# B&R Automation Studio project mappDatabase
Automation Studio 4.9.5.36 SP; technology packages: mapp 5.16.1, mappView 5.16.1

## Configuration Config1

CPU PC_any, AutomationRuntime E4.90, Build 4.1.2, Safety 0.0, Vc V4.45.0

### Task classes (Cpu.sw)
```
Cyclic#1 (cycle 10000 us):
  mappDB <- mappDatabase.mappDB.prg
  RecipeSamp <- mappDatabase.RecipeSample.prg
Binaries: mvLoader, udbdef, arsvcreg, TCData, arconfig, User, Role, Config, iomap, asfw, ashwac, ashwd, sysconf
Libraries: MpDatabase, MpBase, AsHttp, runtime, MpCom, AsBrStr, astime, arssl, asieccon, fileio, standard, IecCheck, sys_lib
```

### Hardware
```
PC : PC_any v1.1.1.0 (OrderNumber=PC)
  ConfigurationID = mappViewSample_Config1
  Cyclic1Duration = 10000
  FileDevice1
  FileDeviceName1 = MpCfgDev
  FileDevicePath1 = C:\Temp
  ActivateOpcUa = 1
  OpcUaInformationModels_PV_Version = 1
```

### Config.mpdatabasecore - PC/mappServices/Config.mpdatabasecore
```
Element gDatabaseCore (Type=mpdatabasecore)
  mapp.Database.Core:
    Name = BrDatabase
    UserName = br
    Password = bandr
    IPAddress  // IPv4 address of the database script
    PortNumber = 85  // SQL port number of the database script
    DBQueries:
      [0]:
        Name = RecipeLoad
        Type:
          Select:
            Columns:
              PV = ::Recipe.DATA
          From = dbo.BrTable
          Where:
            [0]:
              Column = product_name
              Operator = eq
              CompareTo:
                Value = {&pv[Recipe.PAR.RecipeName]}
      [1]:
        Name = RecipeSave
        Type = UPDATE
          TableName = dbo.BrTable
          Columns:
            PV = ::Recipe.DATA
          Where:
            [0]:
              Column = product_name
              Operator = eq
              CompareTo:
                Value = {&pv[Recipe.PAR.RecipeName]}
      [2]:
        Name = RecipeDelete
        Type = DELETE
          TableName = dbo.BrTable
          Where:
            [0]:
              Column = product_name
              Operator = eq
              CompareTo:
                Value = {&pv[Recipe.PAR.RecipeName]}
      [3]:
        Name = RecipeNew
        Type = INSERT
          Into = dbo.BrTable
          Columns:
            PV = ::Recipe.DATA
      [4]:
        Name = RecipeList
        Type = Custom
          Query = SELECT product_name FROM dbo.BrTable WHERE product_name LIKE '%'
          Columns = SingleColumns
            [0]:
              Column = product_name
              PV = ::Recipe.PAR.RecipeName
```

## Logical view

Binary libraries used (declarations not repeated): operator, runtime, astime, AsIecCon, AsHttp, AsBrStr, standard, IecCheck, sys_lib, FileIO, AsICMP, MpCom 5.14.1, MpBase, MpDatabase 5.16.1

### Package Logical/Libraries - Global libraries

### Library Logical/Libraries/MpCfg (IEC)

#### Types.typ - Exported data types
```iecst
TYPE
	MpCfgInfoType : 	STRUCT
		state : MpCfgStateType;
		DevLink_1 : DevLink;
		FileOpen_1 : FileOpen;
		FileRead_1 : FileRead;
		FileWrite_1 : FileWrite;
		FileClose_1 : FileClose;
		MpComConfigManager_1 : MpComConfigManager;
		Buffer : ARRAY[0..MpCfgMaxBufferSize]OF USINT;
		DataOffset1 : DINT;
		DataOffset2 : DINT;
		DataOffset3 : DINT;
		DataLen : DINT;
		FileLen : DINT;
		tmpStr1 : STRING[MpCfgMaxNameSize];
		tmpStr2 : STRING[MpCfgMaxNameSize];
		idx : UDINT;
	END_STRUCT;
	MpCfgStateType :
		(
		stateWait,
		stateDevLink,
		stateExport,
		stateOpen,
		stateRead,
		stateWrite,
		stateClose,
		stateFindGroup,
		stateFindData,
		stateInsertData,
		stateImport,
		stateError
		);
	MpCfgGroupArray : 	STRUCT
		Item : ARRAY[0..9]OF STRING[MpCfgMaxNameSize];
	END_STRUCT;
END_TYPE
```

#### Constants.var - Exported constants
```iecst
(*Buffer and variable sizes*)
VAR CONSTANT
	MpCfgMaxBufferSize : UINT := 20000; (*Maximum size of the configuration file*)
	MpCfgMaxNameSize : UINT := 200; (*Maximum length of the parameter name*)
	MpCfgMaxValueSize : UINT := 200; (*Maximum length of the value information*)
END_VAR
(*Error numbers*)
VAR CONSTANT
	MpCfgBufferSizeExceeded : DINT := 10001; (*Configuration file is larger than MpCfgMaxBufferSize | Increase value of MpCfgMaxBufferSize*)
	MpCfgDataTypeSizeExceeded : DINT := 10002; (*Data type information is larger than MpCfgMaxNameSize | Increase value of MpCfgMaxNameSize*)
	MpCfgValueSizeExceeded : DINT := 10003; (*Value length is larger than MpCfgMaxNameSize | Increase value of MpCfgMaxNameSize*)
	MpCfgGroupNotFound0 : DINT := 10010; (*Group name does not exist | Check group array data at index x*)
	MpCfgGroupNotFound1 : DINT := 10011; (*Group name does not exist | Check group array data at index x*)
	MpCfgGroupNotFound2 : DINT := 10012; (*Group name does not exist | Check group array data at index x*)
	MpCfgGroupNotFound3 : DINT := 10013; (*Group name does not exist | Check group array data at index x*)
	MpCfgGroupNotFound4 : DINT := 10014; (*Group name does not exist | Check group array data at index x*)
	MpCfgGroupNotFound5 : DINT := 10015; (*Group name does not exist | Check group array data at index x*)
	MpCfgGroupNotFound6 : DINT := 10016; (*Group name does not exist | Check group array data at index x*)
	MpCfgGroupNotFound7 : DINT := 10017; (*Group name does not exist | Check group array data at index x*)
	MpCfgGroupNotFound8 : DINT := 10018; (*Group name does not exist | Check group array data at index x*)
	MpCfgGroupNotFound9 : DINT := 10019; (*Group name does not exist | Check group array data at index x*)
	MpCfgParaNotFound : DINT := 10020; (*Parameter name does not exist in configuration | Double check parameter name*)
	MpCfgTypeNotFound : DINT := 10021; (*Data type information was not found | Shouldnt happen but just in case it does*)
	MpCfgValueNotFound : DINT := 10022; (*Value information was not found | Shouldnt happen but just in case it does*)
	MpCfgParaNameEmpty : DINT := 10030; (*Parameter name is empty*)
	MpCfgMpLinkEmpty : DINT := 10031; (*mapp Link is missing*)
END_VAR
(*Read/Write constants*)
VAR CONSTANT
	MpCfgRead : BOOL := FALSE;
	MpCfgWrite : BOOL := TRUE;
END_VAR
```

#### MpCfg.fun - Exported functions and function blocks
```iecst
FUNCTION_BLOCK MpCfgRW
	VAR_INPUT
		MpLink : {REDUND_UNREPLICABLE} MpComIdentType;
		Enable : BOOL;
		ReadWrite : BOOL;
		ErrorReset : BOOL;
		ParaName : STRING[MpCfgMaxNameSize];
		ParaValue : STRING[MpCfgMaxValueSize];
		GroupArray : REFERENCE TO MpCfgGroupArray;
	END_VAR
	VAR_OUTPUT
		Active : BOOL;
		Error : BOOL;
		StatusID : DINT;
		CommandDone : BOOL;
		DataType : STRING[50];
		Value : STRING[MpCfgMaxValueSize];
	END_VAR
	VAR
		Info : MpCfgInfoType;
		zzEdge00000 : BOOL;
		zzEdge00001 : BOOL;
	END_VAR
END_FUNCTION_BLOCK

FUNCTION FindInMem : DINT
	VAR_INPUT
		data1 : UDINT;
		len1 : UDINT;
		data2 : UDINT;
		len2 : UDINT;
		direction : BOOL;
	END_VAR
	VAR
		idx : UDINT;
	END_VAR
END_FUNCTION
```

#### MpCfg.st
```iecst
// -------------------------------------------------------------------------
// Read mapp configuration parameter
// -------------------------------------------------------------------------
FUNCTION_BLOCK MpCfgRW
	// Abort command
	IF EDGENEG(Enable) THEN
		// Close file if it was already opened
		IF Info.state >= stateOpen AND Info.state <> stateError THEN
			Info.state := stateClose;
		END_IF
	END_IF

	// -------------------------------------------------------------------------
	// MpLink state machine
	CASE Info.state OF
		// -------------------------------------------------------------------------
		// Wait for new command
		stateWait:
			// Reset all funtion blocks
			Info.DevLink_1.enable 				:= FALSE;
			Info.DevLink_1();
			Info.MpComConfigManager_1.Enable 	:= FALSE;
			Info.MpComConfigManager_1();
			Info.FileOpen_1.enable				:= FALSE;
			Info.FileOpen_1();
			Info.FileRead_1.enable				:= FALSE;
			Info.FileRead_1();
			Info.FileClose_1.enable				:= FALSE;
			Info.FileClose_1();

			// New command
			IF EDGEPOS(Enable) THEN
				// Make sure MpLink is not empty
				IF MpLink.Internal[0] = 0 THEN
					StatusID := MpCfgMpLinkEmpty;
					Info.state := stateError;
				ELSE
					// Make sure parameter is not empty
					IF ParaName = '' THEN
						StatusID := MpCfgParaNameEmpty;
						Info.state := stateError;
					ELSE
						// Set start values
						Active := TRUE;
						DataType := '';
						Value := '';
						brsmemset(ADR(Info.Buffer), 0, SIZEOF(Info.Buffer));
						Info.state := stateDevLink;
					END_IF
				END_IF
			ELSE
				IF NOT Enable THEN
					CommandDone := FALSE;
				END_IF
				Active := FALSE;
			END_IF
			// -------------------------------------------------------------------------
		// Link file device used for exporting data
		stateDevLink:
			Info.DevLink_1.enable 	:= TRUE;
			Info.DevLink_1.pDevice	:= ADR('MpCfgDev');
			Info.DevLink_1.pParam	:= ADR('/DEVICE=C:/');
			Info.DevLink_1();

			// Success
			IF Info.DevLink_1.status = ERR_OK OR Info.DevLink_1.status = fiERR_DEVICE_ALREADY_EXIST THEN
				Info.state := stateExport;
			// Errror
			ELSIF Info.DevLink_1.status <> ERR_FUB_BUSY THEN
				StatusID := Info.DevLink_1.status;
				Info.state := stateError;
			END_IF
		// -------------------------------------------------------------------------
		// Export mapp data
		stateExport:
			Info.MpComConfigManager_1.Enable 		:= TRUE;
			Info.MpComConfigManager_1.MpLink		:= ADR(MpLink);
			Info.MpComConfigManager_1.DeviceName 	:= ADR('MpCfgDev');
			Info.MpComConfigManager_1.FileName 		:= ADR('MpCfg.xml');
			Info.MpComConfigManager_1.Scope			:= mpCOM_CONFIG_SCOPE_COMPONENT;
			Info.MpComConfigManager_1.Export		:= TRUE;
			Info.MpComConfigManager_1.Import		:= FALSE;
			Info.MpComConfigManager_1();

			// Success
			IF Info.MpComConfigManager_1.CommandDone AND NOT Info.MpComConfigManager_1.Error THEN
				Info.state := stateOpen;
			// Errror
			ELSIF Info.MpComConfigManager_1.Error THEN
				StatusID := Info.MpComConfigManager_1.StatusID;
				Info.state := stateError;
			END_IF
		// -------------------------------------------------------------------------
		// Open mapp data
		stateOpen:
			Info.FileOpen_1.enable		:= TRUE;
			Info.FileOpen_1.pDevice 	:= ADR('MpCfgDev');
			Info.FileOpen_1.pFile		:= ADR('MpCfg.xml');
			Info.FileOpen_1.mode 		:= fiREAD_WRITE;
			Info.FileOpen_1();

			// Success
			IF Info.FileOpen_1.status = ERR_OK THEN
				IF Info.FileOpen_1.filelen > SIZEOF(Info.Buffer) THEN
					StatusID := MpCfgBufferSizeExceeded;
					Info.state := stateError;
				ELSE
					Info.state := stateRead;
				END_IF
			// Errror
			ELSIF Info.FileOpen_1.status <> ERR_FUB_BUSY THEN
				StatusID := Info.FileOpen_1.status;
				Info.state := stateError;
			END_IF

		// -------------------------------------------------------------------------
		// Read mapp data file
		stateRead:
			Info.FileRead_1.enable		:= TRUE;
			Info.FileRead_1.ident		:= Info.FileOpen_1.ident;
			Info.FileRead_1.len			:= Info.FileOpen_1.filelen;
			Info.FileRead_1.pDest		:= ADR(Info.Buffer);
			Info.FileRead_1();

			// Success
			IF Info.FileRead_1.status = ERR_OK THEN
				Info.idx := 0;
				Info.DataOffset1 := 0;
				// Find group id first
				IF ADR(GroupArray) <> 0 THEN
					// Make sure array has at least one entry
					IF GroupArray.Item[0] <> '' THEN
						Info.state := stateFindGroup;
					// Find unique parameter
					ELSE
						Info.state := stateFindData;
					END_IF
				// Find unique parameter
				ELSE
					Info.state := stateFindData;
				END_IF
			// Errror
			ELSIF Info.FileRead_1.status <> ERR_FUB_BUSY THEN
				StatusID := Info.FileRead_1.status;
				Info.state := stateError;
			END_IF

		// -------------------------------------------------------------------------
		// Write mapp data file
		stateWrite:
			Info.FileWrite_1.enable		:= TRUE;
			Info.FileWrite_1.ident		:= Info.FileOpen_1.ident;
			Info.FileWrite_1.len		:= Info.FileLen;
			Info.FileWrite_1.pSrc		:= ADR(Info.Buffer);
			Info.FileWrite_1();

			// Success
			IF Info.FileWrite_1.status = ERR_OK THEN
				Info.state := stateClose;
			// Errror
			ELSIF Info.FileWrite_1.status <> ERR_FUB_BUSY THEN
				StatusID := Info.FileWrite_1.status;
				Info.state := stateError;
			END_IF

		// -------------------------------------------------------------------------
		// Find group data
		stateFindGroup:
			// Prepare group string
			Info.tmpStr1 := '<Group ID="';
			brsstrcat(ADR(Info.tmpStr1), ADR(GroupArray.Item[Info.idx]));
			brsstrcat(ADR(Info.tmpStr1), ADR('"'));
			// Find property string
			Info.DataOffset1 := Info.DataOffset1+FindInMem(ADR(Info.Buffer)+Info.DataOffset1, Info.FileOpen_1.filelen, ADR(Info.tmpStr1), brsstrlen(ADR(Info.tmpStr1)), FALSE);

			// Found group string
			IF Info.DataOffset1 > -1 THEN
				// Find next group name
				IF Info.idx < SIZEOF(GroupArray)/SIZEOF(GroupArray.Item[0]) THEN
					Info.idx := Info.idx + 1;
					IF GroupArray.Item[Info.idx] = '' THEN
						Info.state := stateFindData;
					END_IF
				// Group was not found
				ELSE
					StatusID := MpCfgGroupNotFound0+Info.idx;
					Info.state := stateError;
				END_IF
			// Group was not found
			ELSE
				StatusID := MpCfgGroupNotFound0+Info.idx;
				Info.state := stateError;
			END_IF
		// -------------------------------------------------------------------------
		// Find data
		stateFindData:
			// Prepare property string
			Info.tmpStr1 := '<Property ID="';
			brsstrcat(ADR(Info.tmpStr1), ADR(ParaName));
			brsstrcat(ADR(Info.tmpStr1), ADR('"'));
			// Find property string
			Info.DataOffset2 := FindInMem(ADR(Info.Buffer)+Info.DataOffset1, Info.FileOpen_1.filelen, ADR(Info.tmpStr1), brsstrlen(ADR(Info.tmpStr1)), FALSE);

			// Found parameter string
			IF Info.DataOffset2 > -1 THEN
				Info.DataOffset1 := Info.DataOffset1+Info.DataOffset2;
				// Prepare data type start string
				Info.tmpStr1 := 'DataType="';
				// Find data type string start
				Info.DataOffset2 := brsstrlen(ADR(Info.tmpStr1))+FindInMem(ADR(Info.Buffer)+Info.DataOffset1, Info.FileOpen_1.filelen, ADR(Info.tmpStr1), brsstrlen(ADR(Info.tmpStr1)), FALSE);

				// Found data type start
				IF Info.DataOffset2 > -1 THEN
					// Prepare data type end string
					Info.tmpStr1 := '"';
					// Find data type string
					Info.DataLen := FindInMem(ADR(Info.Buffer)+Info.DataOffset1+Info.DataOffset2, Info.FileOpen_1.filelen, ADR(Info.tmpStr1), brsstrlen(ADR(Info.tmpStr1)), FALSE);

					// Found data type end, copy data to output
					IF Info.DataLen > -1 THEN
						brsmemset(ADR(DataType), 0, SIZEOF(DataType));
						brsmemcpy(ADR(DataType), ADR(Info.Buffer)+Info.DataOffset1+Info.DataOffset2, Info.DataLen);

						// Prepare value start string
						Info.tmpStr1 := 'Value="';
						// Find data type string start
						Info.DataOffset2 := brsstrlen(ADR(Info.tmpStr1))+FindInMem(ADR(Info.Buffer)+Info.DataOffset1, Info.FileOpen_1.filelen, ADR(Info.tmpStr1), brsstrlen(ADR(Info.tmpStr1)), FALSE);

						// Found value start
						IF Info.DataOffset2 > -1 THEN
							// Prepare value end string
							Info.tmpStr1 := '"';
							// Find value end string
							Info.DataLen := FindInMem(ADR(Info.Buffer)+Info.DataOffset1+Info.DataOffset2, Info.FileOpen_1.filelen, ADR(Info.tmpStr1), brsstrlen(ADR(Info.tmpStr1)), FALSE);

							// Found value end, copy data to output
							IF Info.DataLen > -1 THEN
								brsmemset(ADR(Value), 0, SIZEOF(Value));
								brsmemcpy(ADR(Value), ADR(Info.Buffer)+Info.DataOffset1+Info.DataOffset2, Info.DataLen);

								// Finish when command is reading
								IF ReadWrite = MpCfgRead THEN
									Info.state := stateClose;
								// Insert new data in next step
								ELSE
									Info.state := stateInsertData;
								END_IF
							// Value end was not found
							ELSE
								StatusID := MpCfgValueNotFound;
								Info.state := stateError;
							END_IF
						// Value start was not found
						ELSE
							StatusID := MpCfgValueNotFound;
							Info.state := stateError;
						END_IF
					// Data type end was not found
					ELSE
						StatusID := MpCfgTypeNotFound;
						Info.state := stateError;
					END_IF
				// Data type end was not found
				ELSE
					StatusID := MpCfgTypeNotFound;
					Info.state := stateError;
				END_IF
			// Parameter name was not found
			ELSE
				StatusID := MpCfgParaNotFound;
				Info.state := stateError;
			END_IF

		// -------------------------------------------------------------------------
		// Insert new data
		stateInsertData:
			// Calculate start address for value
			Info.DataOffset3 := ADR(Info.Buffer)+Info.DataOffset1+Info.DataOffset2;
			// Calculate remaining data
			Info.DataLen := Info.FileOpen_1.filelen-(Info.DataOffset1+Info.DataOffset2);

			brsmemmove(Info.DataOffset3+brsstrlen(ADR(ParaValue)), Info.DataOffset3+brsstrlen(ADR(Value)), Info.DataLen-brsstrlen(ADR(Value))+1);
			brsmemcpy(Info.DataOffset3, ADR(ParaValue), brsstrlen(ADR(ParaValue)));

			// New value is shorter than old
			IF brsstrlen(ADR(Value)) >= brsstrlen(ADR(ParaValue)) THEN
				Info.FileLen := Info.FileOpen_1.filelen;
				// Fill taling memory with LF if new data is smaller than old
				brsmemset(ADR(Info.Buffer)+Info.FileLen, 10, brsstrlen(ADR(Value))-brsstrlen(ADR(ParaValue)));
			// New value is larger than old
			ELSE
				Info.FileLen := Info.FileOpen_1.filelen+(brsstrlen(ADR(ParaValue))-brsstrlen(ADR(Value)));
			END_IF

			Info.state := stateWrite;

		// -------------------------------------------------------------------------
		// Close mapp data file
		stateClose:
			Info.FileClose_1.enable		:= TRUE;
			Info.FileClose_1.ident		:= Info.FileOpen_1.ident;
			Info.FileClose_1();

			// Success
			IF Info.FileClose_1.status = ERR_OK THEN
				Info.FileOpen_1.enable := FALSE;

				// When we read it ends here
				IF ReadWrite = MpCfgRead THEN
					Active := FALSE;
					CommandDone := TRUE;
					Info.state := stateWait;
				// Import new configuration
				ELSE
					Info.state := stateImport;
				END_IF
				// Errror
			ELSIF Info.FileClose_1.status <> ERR_FUB_BUSY THEN
				StatusID := Info.FileClose_1.status;
				Info.state := stateError;
			END_IF

		// -------------------------------------------------------------------------
		// Import mapp data
		stateImport:
			Info.MpComConfigManager_1.Enable 		:= TRUE;
			Info.MpComConfigManager_1.MpLink		:= ADR(MpLink);
			Info.MpComConfigManager_1.DeviceName 	:= ADR('MpCfgDev');
			Info.MpComConfigManager_1.FileName 		:= ADR('MpCfg.xml');
			Info.MpComConfigManager_1.Scope			:= mpCOM_CONFIG_SCOPE_COMPONENT;
			Info.MpComConfigManager_1.Export		:= FALSE;
			Info.MpComConfigManager_1.Import		:= TRUE;
			Info.MpComConfigManager_1();

			// Success
			IF Info.MpComConfigManager_1.CommandDone AND NOT Info.MpComConfigManager_1.Error THEN
				Active := FALSE;
				CommandDone := TRUE;
				Info.state := stateWait;
			// Errror
			ELSIF Info.MpComConfigManager_1.Error THEN
				StatusID := Info.MpComConfigManager_1.StatusID;
				Info.state := stateError;
			END_IF

		// -------------------------------------------------------------------------
		// Error state
		stateError:
			// Close file when it is open
			IF Info.FileOpen_1.enable THEN
				Info.FileClose_1.enable	:= TRUE;
				Info.FileClose_1.ident	:= Info.FileOpen_1.ident;
				Info.FileClose_1();
			END_IF

			// Set flags
			Active := FALSE;
			Error := TRUE;
			CommandDone := TRUE;

			// Wait for error reset
			IF ErrorReset THEN
				StatusID := 0;
				Error := FALSE;
				Info.state := stateWait;
			END_IF
	END_CASE;

	ErrorReset := FALSE;
END_FUNCTION_BLOCK
```

#### LocalFunctions.st
```iecst
//******************************************************************************************************
// Find second data in first data
//******************************************************************************************************
FUNCTION FindInMem
	FindInMem := -1;
	IF (len1 > len2) THEN
		IF(direction) THEN
			idx := len1 - len2;
			WHILE(idx > 0) DO
				IF (brsmemcmp(data1 + idx, data2, len2) = 0) THEN
					FindInMem := idx;
					EXIT;
				END_IF
				idx := idx - 1;
			END_WHILE;
		ELSE
			FOR idx:=0 TO len1 - len2 DO
				IF (brsmemcmp(data1 + idx, data2, len2) = 0) THEN
					FindInMem := idx;
					EXIT;
				END_IF
			END_FOR;
		END_IF
	END_IF
END_FUNCTION
```

#### changelog.txt
```
Version 1.0 (23.12.2021)
- First public release
```

- Visualisation Logical/mappView (not shown)

### Program Logical/mappDatabase/mappDB (IEC)

#### Main.st - Init, cyclic, exit code
```iecst
PROGRAM _INIT
	// --------------------------------------------------------------------------------------------------------------------
	// Preset function blocks
	MpDatabaseCore_0.MpLink := ADR(gDatabaseCore);
	MpDatabaseQuery_0.MpLink := ADR(gDatabaseCore);

	SqlTimeout.PT := TIMEOUT;

	REPEAT
		MpCfgRW_01.Enable 		:= TRUE;
		MpCfgRW_01.MpLink 		:= gDatabaseCore;
		MpCfgRW_01.ReadWrite 	:= MpCfgRead;
		MpCfgRW_01.ParaName 	:= 'IPAddress';
		MpCfgRW_01.GroupArray	:= 0;
		MpCfgRW_01();
		UNTIL MpCfgRW_01.CommandDone
	END_REPEAT;

END_PROGRAM

PROGRAM _CYCLIC
		// Trigger ping request
	PingTimer.IN := TRUE;
	PingTimer.PT := PING_TIMEOUT;
	PingTimer();
	// Try to ping network share if not connected
	IF(MpCfgRW_01.Value <> '' AND PingTimer.Q) THEN
		IcmpPing_0(enable := 1, pHost := ADR(MpCfgRW_01.Value), timeout := PING_TIMEOUT);
		// Ping was OK
		IF(IcmpPing_0.status = ERR_OK) THEN
			PingTimer(IN := FALSE);
			Database.PAR.CanPing := TRUE;
			// Disconnect from share when ping failed
		ELSIF(IcmpPing_0.status <> ERR_FUB_BUSY) THEN
			PingTimer(IN := FALSE);
			Database.PAR.CanPing := FALSE;
			IF(Database.PAR.IsConnected) THEN
				Database.CMD.Disconnect := TRUE;
			END_IF
		END_IF
	ELSIF(PingTimer.Q) THEN
		PingTimer(IN := FALSE);
	END_IF

	// --------------------------------------------------------------------------------------------------------------------
	// Database state machine
	// --------------------------------------------------------------------------------------------------------------------
	CASE dbState OF
		// --------------------------------------------------------------------------------------------------------------------
		// Wait state
		dbSTATE_WAIT:
			// --------------------------------------------------------------------------------------------------------------------
			// Connect to database
			IF Database.CMD.Connect THEN
				dbState := dbSTATE_CONNECT;
			END_IF

			// Disconnect from database
			IF Database.CMD.Disconnect THEN
				dbState := dbSTATE_DISCONNECT;
			END_IF

			// Execute SQL command
			IF Database.CMD.Execute THEN
				dbState := dbSTATE_QUERY;
			END_IF

			// Get next entry
			IF Database.CMD.NextRow THEN
				dbState := dbSTATE_NEXT;
			END_IF

			// --------------------------------------------------------------------------------------------------------------------
			// Reset error information and timeout timer
			IF Database.CMD.Connect OR Database.CMD.Disconnect OR Database.CMD.Execute OR Database.CMD.NextRow THEN
				Database.ERR.No := 0;
				brsmemset(ADR(Database.ERR.Text), 0, SIZEOF(Database.ERR.Text));

				MpDatabaseCore_0.Enable := TRUE;
				MpDatabaseQuery_0.Enable := TRUE;
				MpDatabaseQuery_0.ErrorReset := TRUE;
				MpDatabaseCore_0.ErrorReset := TRUE;
				MpDatabaseQuery_0();
				MpDatabaseCore_0();

				SqlTimeout.IN := 0;
				SqlTimeout();
			END_IF

		// --------------------------------------------------------------------------------------------------------------------
		// Connect state
		dbSTATE_CONNECT:
			SqlTimeout.IN := 1;
			SqlTimeout();

			IF MpDatabaseCore_0.CommandDone OR MpDatabaseCore_0.Error THEN
				IF MpDatabaseCore_0.Error THEN
					Database.ERR.No := MpDatabaseCore_0.StatusID;
					dbState := dbSTATE_ERROR;
				ELSE
					Database.CMD.Connect := FALSE;
					dbState := dbSTATE_WAIT;
				END_IF
			ELSIF SqlTimeout.Q THEN
				Database.ERR.No := ERR_SQL_TIMEOUT_CONNECT;
				MpDatabaseCore_0.Enable := FALSE;
				dbState := dbSTATE_ERROR;
			END_IF

		// --------------------------------------------------------------------------------------------------------------------
		// Disconnect state
		dbSTATE_DISCONNECT:
			SqlTimeout.IN := 1;
			SqlTimeout();

			IF MpDatabaseCore_0.CommandDone OR MpDatabaseCore_0.Error THEN

				IF MpDatabaseCore_0.Error THEN
					Database.ERR.No := MpDatabaseCore_0.StatusID;
					dbState := dbSTATE_ERROR;
				ELSE
					Database.CMD.Disconnect := FALSE;
					dbState := dbSTATE_WAIT;
				END_IF
			ELSIF SqlTimeout.Q THEN
				Database.ERR.No := ERR_SQL_TIMEOUT_CONNECT;
				MpDatabaseCore_0.Enable := FALSE;
				dbState := dbSTATE_ERROR;
			END_IF

		// --------------------------------------------------------------------------------------------------------------------
		// Query state
		dbSTATE_QUERY:
			SqlTimeout.IN := 1;
			SqlTimeout();

			IF MpDatabaseQuery_0.CommandDone OR MpDatabaseQuery_0.Error THEN
				Database.CMD.Execute := FALSE;

				IF MpDatabaseQuery_0.Error THEN
					Database.ERR.No := MpDatabaseQuery_0.StatusID;
					dbState := dbSTATE_ERROR;
				ELSE
					dbState := dbSTATE_WAIT;
				END_IF
			ELSIF NOT Database.PAR.IsConnected THEN
				Database.ERR.No := ERR_SQL_NOT_CONNECTED;
				dbState := dbSTATE_ERROR;
			ELSIF SqlTimeout.Q THEN
				Database.ERR.No := ERR_SQL_TIMEOUT_QUERY;
				MpDatabaseQuery_0.Enable := FALSE;
				dbState := dbSTATE_ERROR;
			END_IF

		// --------------------------------------------------------------------------------------------------------------------
		// Read next row
		dbSTATE_NEXT:
			SqlTimeout.IN := 1;
			SqlTimeout();

			IF MpDatabaseQuery_0.CommandDone OR MpDatabaseQuery_0.Error THEN
				Database.CMD.NextRow := FALSE;

				IF MpDatabaseQuery_0.Error THEN
					Database.ERR.No := MpDatabaseQuery_0.StatusID;
					dbState := dbSTATE_ERROR;
				ELSE
					dbState := dbSTATE_WAIT;
				END_IF
			ELSIF SqlTimeout.Q THEN
				Database.ERR.No := ERR_SQL_TIMEOUT_QUERY;
				MpDatabaseQuery_0.Enable := FALSE;
				dbState := dbSTATE_ERROR;
			END_IF

		// --------------------------------------------------------------------------------------------------------------------
		// Error state
		dbSTATE_ERROR:
			Database.CMD.Connect := FALSE;
			Database.CMD.Disconnect := FALSE;
			Database.CMD.Execute := FALSE;
			Database.CMD.NextRow := FALSE;

			IF Database.ERR.No = mpDATABASE_ERR_SQL_SERVER THEN
				Database.ERR.Text := 'Error response from SQL server. Check SQL syntax!';
			ELSIF Database.ERR.No = mpCOM_ERR_ACTIVATION THEN
				Database.ERR.Text := 'Could not create component query. Try to reboot PLC and script!';
			ELSIF Database.ERR.No = mpDATABASE_ERR_QUERY_RESULT THEN
				Database.ERR.Text := 'Check the query to determine if correct table and column names were used.';
			ELSIF Database.ERR.No = mpDATABASE_INF_NO_DATA THEN
				Database.ERR.Text := 'No more data available.';
			ELSIF Database.ERR.No = mpDATABASE_ERR_HTTP_SERVER AND NOT Database.PAR.IsConnected THEN
				Database.ERR.Text := 'Not connected to database. Try to reboot PLC and script!';
			ELSIF Database.ERR.No = ERR_SQL_TIMEOUT_CONNECT THEN
				Database.ERR.Text := 'SQL timeout during connection. Make sure script and server is running.';
			ELSIF Database.ERR.No = ERR_SQL_TIMEOUT_QUERY THEN
				Database.ERR.Text := 'SQL timeout during query.';
			ELSIF Database.ERR.No = ERR_SQL_NOT_CONNECTED THEN
				Database.ERR.Text := 'Not connected to database. Call command connect first';
			ELSE
				Database.ERR.Text := 'Generic SQL error.';
			END_IF

			dbState := dbSTATE_WAIT;
	END_CASE;

	// --------------------------------------------------------------------------------------------------------------------
	// Function block calls
	IF NOT MpDatabaseQuery_0.ErrorReset THEN
		MpDatabaseQuery_0.Execute := Database.CMD.Execute;
		MpDatabaseQuery_0.Next := Database.CMD.NextRow;
		MpDatabaseQuery_0.Name := ADR(Database.PAR.QueryName);
	END_IF
	MpDatabaseQuery_0();

	IF NOT MpDatabaseCore_0.ErrorReset THEN
		MpDatabaseCore_0.Connect := Database.CMD.Connect;
		MpDatabaseCore_0.Disconnect := Database.CMD.Disconnect;
	END_IF
	MpDatabaseCore_0();

	// Transfer function block data to global structure
	Database.PAR.IsConnected := MpDatabaseCore_0.Connected;
	Database.PAR.RowsTotal := MpDatabaseQuery_0.Info.Rows.Total;
	Database.PAR.RowsRead := MpDatabaseQuery_0.Info.Rows.Read;
	Database.PAR.RowsRemaining := MpDatabaseQuery_0.Info.Rows.Remaining;

	// Clear error reset command
	MpDatabaseQuery_0.ErrorReset := FALSE;
	MpDatabaseCore_0.ErrorReset := FALSE;

END_PROGRAM

PROGRAM _EXIT
	// --------------------------------------------------------------------------------------------------------------------
	// Exit function blocks
	MpDatabaseCore_0.Enable := FALSE;
	MpDatabaseCore_0();

	MpDatabaseQuery_0.Enable := FALSE;
	MpDatabaseQuery_0();

END_PROGRAM
```

#### LocalTypes.typ - Local data types
```iecst
TYPE
	dbState_Enum :
		(
		dbSTATE_WAIT,
		dbSTATE_CONNECT,
		dbSTATE_DISCONNECT,
		dbSTATE_QUERY,
		dbSTATE_NEXT,
		dbSTATE_ERROR
		);
END_TYPE
```

#### LocalVariables.var - Local variables
```iecst
(*------------------------------------------------------------------------------------------------------------------------------------------------------------------------------------------------------------------------*)
(*SQL function calls*)
VAR
	MpDatabaseCore_0 : MpDatabaseCore; (*mappDatabase main function block*)
	MpDatabaseQuery_0 : MpDatabaseQuery; (*mappDatabase query*)
END_VAR
(*------------------------------------------------------------------------------------------------------------------------------------------------------------------------------------------------------------------------*)
(*Local variables*)
VAR
	SqlTimeout : TON_10ms; (*Timeout for SQL commands*)
	dbState : dbState_Enum; (*State machine*)
END_VAR
(*------------------------------------------------------------------------------------------------------------------------------------------------------------------------------------------------------------------------*)
(*Configuration for database managment*)
VAR CONSTANT
	TIMEOUT : UINT := 100; (*Timeout for SQL connection and query, default is 100=>1s*)
END_VAR
(*------------------------------------------------------------------------------------------------------------------------------------------------------------------------------------------------------------------------*)
(*Local constants*)
VAR CONSTANT
	ERR_SQL_TIMEOUT_CONNECT : UINT := 10000; (*Timeout error for SQL connection*)
	ERR_SQL_TIMEOUT_QUERY : UINT := 10001; (*Timeout error for SQL query*)
	ERR_SQL_NOT_CONNECTED : UINT := 10010; (*Can not execute when not connected*)
END_VAR
```

### Program Logical/mappDatabase/RecipeSample (IEC)

#### Main.st - Init, cyclic, exit code
```iecst
PROGRAM _INIT
END_PROGRAM

PROGRAM _CYCLIC

	// Generate a list with all recipe names
	IF EDGEPOS(Database.PAR.IsConnected) THEN
		Recipe.CMD.List := TRUE;
	END_IF
	IF EDGEPOS(Recipe.CMD.List) THEN
		Database.PAR.QueryName := 'RecipeList';
		Database.CMD.Execute := TRUE;
		idx := 0;
		brsmemset(ADR(Recipe.PAR.RecipeNames), 0, SIZEOF(Recipe.PAR.RecipeNames));
	END_IF
	// Translate recipe names to mappView data providers
	IF Recipe.CMD.List AND (EDGENEG(Database.CMD.Execute) OR EDGENEG(Database.CMD.NextRow)) THEN
		brsstrcpy(ADR(Recipe.PAR.RecipeNames[idx]), ADR('{"value":"'));
		brsstrcat(ADR(Recipe.PAR.RecipeNames[idx]), ADR(Recipe.DATA.product_name));
		brsstrcat(ADR(Recipe.PAR.RecipeNames[idx]), ADR('","text":"'));
		brsstrcat(ADR(Recipe.PAR.RecipeNames[idx]), ADR(Recipe.DATA.product_name));
		brsstrcat(ADR(Recipe.PAR.RecipeNames[idx]), ADR('"}'));

		// Read next entry as long as we have entries and space
		IF Database.PAR.RowsRemaining > 0 AND idx < SIZEOF(Recipe.PAR.RecipeNames)/SIZEOF(Recipe.PAR.RecipeNames[idx]) THEN
			idx := idx + 1;
			Database.CMD.NextRow := TRUE;
		ELSE
			Recipe.CMD.List := FALSE;
		END_IF
	END_IF

	// Load recipe
	IF Recipe.CMD.Load THEN
		// Reset command
		IF EDGENEG(Database.CMD.Execute) THEN
			Recipe.CMD.Load := FALSE;
		// Trigger database command
		ELSE
			Database.PAR.QueryName := 'RecipeLoad';
			Database.CMD.Execute := TRUE;
		END_IF
	END_IF

	// Save recipe
	IF Recipe.CMD.Save OR Recipe.CMD.Rename THEN
		// Reset command
		IF EDGENEG(Database.CMD.Execute) THEN
			Recipe.CMD.Save := FALSE;
			IF Recipe.CMD.Rename THEN
				Recipe.CMD.Rename := FALSE;
				Recipe.CMD.List := TRUE;
			END_IF
		// Trigger database command
		ELSE
			Database.PAR.QueryName := 'RecipeSave';
			Database.CMD.Execute := TRUE;
		END_IF
	END_IF

	// New recipe
	IF Recipe.CMD.New THEN
		// Reset command
		IF EDGENEG(Database.CMD.Execute) THEN
			Recipe.CMD.New := FALSE;
			Recipe.CMD.List := TRUE;
		// Trigger database command
		ELSE
			Database.PAR.QueryName := 'RecipeNew';
			Database.CMD.Execute := TRUE;
		END_IF
	END_IF

	// Delete recipe
	IF Recipe.CMD.Delete THEN
		// Reset command
		IF EDGENEG(Database.CMD.Execute) THEN
			Recipe.CMD.Delete := FALSE;
			Recipe.CMD.List := TRUE;
		// Trigger database command
		ELSE
			Database.PAR.QueryName := 'RecipeDelete';
			Database.CMD.Execute := TRUE;
		END_IF
	END_IF

END_PROGRAM
```

#### LocalVariables.var - Local variables
```iecst
VAR
	idx : USINT;
END_VAR
```

### dbTypes.typ
```iecst
TYPE
	dbCMD : 	STRUCT  (*Database command structure*)
		Connect : BOOL; (*Connect to database*)
		Disconnect : BOOL; (*Disconnect from database*)
		Execute : BOOL; (*Execute SQL command*)
		NextRow : BOOL; (*Get next response row*)
	END_STRUCT;
	dbPAR : 	STRUCT  (*Database parameter structure*)
		IsConnected : BOOL; (*Shows if database connection is active*)
		QueryName : STRING[200]; (*Name of the SQL query define under mappServices*)
		RowsTotal : UDINT; (*Total number of response rows*)
		RowsRead : UDINT; (*Rows already reqeusted*)
		RowsRemaining : UDINT; (*Rows remaining*)
	END_STRUCT;
	dbERR : 	STRUCT  (*Database error structure*)
		Text : STRING[200]; (*Error text*)
		No : DINT; (*Error number*)
	END_STRUCT;
	dbMAIN : 	STRUCT  (*Database main structure*)
		CMD : dbCMD;
		PAR : dbPAR;
		ERR : dbERR;
	END_STRUCT;
	recCMD : 	STRUCT  (*Recipe command structure*)
		Load : BOOL; (*Load recipe*)
		Save : BOOL; (*Save recipe*)
		New : BOOL; (*Create new recipe*)
		Delete : BOOL; (*Delete recipe*)
		Rename : BOOL; (*Rename recipe*)
		List : BOOL; (*Get list of all recipes*)
	END_STRUCT;
	recPAR : 	STRUCT  (*Recipe parameter structure*)
		RecipeNames : ARRAY[0..9]OF STRING[200]; (*List of all recipes formated for mappView*)
		RecipeName : STRING[200]; (*Current recipe name for command*)
	END_STRUCT;
	recDATA : 	STRUCT  (*Recipe data structure*)
		product_name : STRING[80];
		sugar : UINT;
		water : UINT;
		milk : UINT;
		temperature : REAL;
	END_STRUCT;
	recMAIN : 	STRUCT  (*Recipe main structure*)
		CMD : recCMD;
		PAR : recPAR;
		DATA : recDATA;
	END_STRUCT;
END_TYPE
```

### dbVariables.var
```iecst
VAR
	Database : dbMAIN; (*Database main structure*)
	Recipe : recMAIN; (*Recipe sample structure*)
END_VAR
```

### changelog.txt
```
Version 1.0 (18.08.2021)
- PythonScript: Added more and detailed debug output
- PythonScript: Added more and detailed error messages
- PythonScript: Print all SQL queries and server response details
- PythonScript: Trim data type string when reading from database
- PythonScript: Change MsSQL database provider to 'ODBC Driver 17 for SQL Server' to support linux systems
- PythonScript: Removed dependecy from MySql driver for data conversion. Removed dependecy from MySql driver for data conversion. It is no longer required to install MySQL driver when using MsSQL.
```

### Program Logical/mappDatabase/test

#### Variables.var
```iecst
VAR
	tmpSTR1 : STRING[80];
	tmpSTR2 : STRING[80];
	create : UINT;
END_VAR
```

#### Main.st
```iecst
PROGRAM _INIT
	(* Insert code here *)

END_PROGRAM

PROGRAM _CYCLIC
	IF create > 0 AND NOT Recipe.CMD.New THEN
		tmpSTR1 := 'TestProduct';
		brsitoa(create, ADR(tmpSTR2));
		brsstrcat(ADR(tmpSTR1), ADR(tmpSTR2));
		Recipe.DATA.product_name := tmpSTR1;
		Recipe.DATA.water := create;
		Recipe.DATA.milk := create;
		Recipe.DATA.sugar := create;
		Recipe.DATA.temperature := create/3.14;
		Recipe.DATA.test1 := UINT_TO_BOOL(create);
		Recipe.DATA.test2 := UINT_TO_SINT(create);
		Recipe.DATA.test3 := UINT_TO_INT(create);
		Recipe.DATA.test4 := UINT_TO_DINT(create);
		Recipe.DATA.test5 := UINT_TO_USINT(create);
		Recipe.DATA.test6 := create;
		Recipe.DATA.test7 := UINT_TO_UDINT(create);
		Recipe.DATA.test8 := UINT_TO_TIME(create);
		Recipe.DATA.test9 := UINT_TO_REAL(create);
		Recipe.DATA.test10 := UINT_TO_LREAL(create);
		Recipe.DATA.test11 := UINT_TO_DATE(create);
		Recipe.DATA.test12 := UINT_TO_DT(create);

		create := create - 1;
		Recipe.CMD.New := TRUE;
	END_IF

END_PROGRAM
```

Listed in the project but not available here: Logical/Global.typ, Logical/Global.var
